Staubli VAL3: Init.pgx

program Init()
  local num l_ni
begin
  //
  nPage=0
  for l_ni=0 to 7
    sMsg[l_ni]=""
  endFor
  //
  nSize=size(A130:ptRoutingPath)
  resize(sList,1,nSize)
  //
  //

  //
  bUserRefresh=bListRefresh=true
  //
  bExit=false

  //
  if bInit
    call JTP()
    libSave()
  endIf
  fFrmTemp.trsf=frmaster.trsf
end
